// TwinCAT 3 PLC project MAS418_PLC
// ProgramVersion: 3.1.4023.0
// libraries:
//   Tc2_Standard, * (Beckhoff Automation GmbH)
//   Tc2_System, * (Beckhoff Automation GmbH)
//   Tc3_Module, * (Beckhoff Automation GmbH)
// project tree:
//   / GlobalTextList.TcGTLO, PlcTask.TcTTO, Visualization Manager.TcVMO (not stored)
//   POUs/ MAIN.TcPOU
//   VISUs/ HMI.TcVIS
// real-time tasks:
//   TASK PlcTask: cycle T#10ms, priority 20, ADS port 350

CONFIGURATION MAS418_PLC
    RESOURCE PLC ON TwinCAT3
        TASK PlcTask(INTERVAL := T#10ms, PRIORITY := 20);
        PROGRAM MAIN WITH PlcTask : MAIN;
    END_RESOURCE
END_CONFIGURATION

// ---- POUs/MAIN.TcPOU
PROGRAM MAIN
VAR
	bEnable : BOOL;
	bStart : BOOL;
	nINT : INT := -32768;
	nUINT : UINT := 65535;
	fREAL : REAL := 255.255;
END_VAR

bEnable := bStart;

END_PROGRAM

// ---- GlobalTextList.TcGTLO
TEXTLIST GlobalTextList
  775 = 'BOOL'
  109 = 'BOOL%i'
  173 = 'DataTypeTesting'
  74 = 'INT'
  710 = 'INT%i'
  986 = 'Power ON'
  573 = 'REAL'
  369 = 'REAL%i'
  65 = 'STRING'
  563 = 'STRING%i'
  393 = 'UINT'
  128 = 'UINT%i'
END_TEXTLIST

// ---- VISUs/HMI.TcVIS
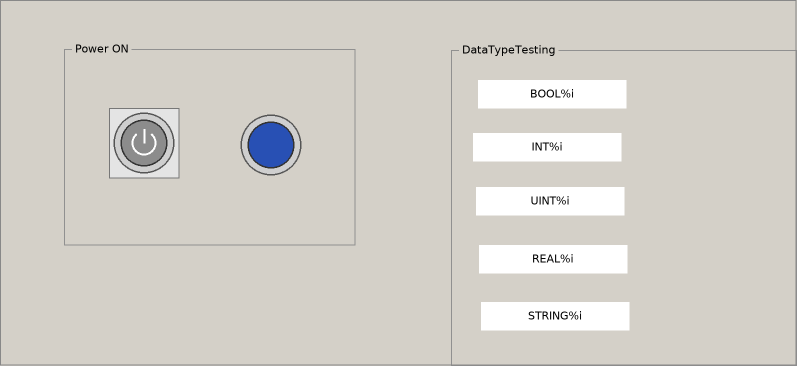
VISUALIZATION HMI  // 797x366
    GroupBox (64,41 291x204), "Power ON"
        PowerSwitch (45,67 70x70), variable: MAIN.bStart, behaviour: TOGGLE, style: Switch-PowerSwitch-Gray
        Lamp1 (172,69 70x70), variable: MAIN.bEnable, style: Lamp-Lamp1-Blue
    GroupBox (451,42 346x324), "DataTypeTesting"
        Textfield (26,37 150x30), "BOOL%i", text variable: MAIN.bEnable
        Textfield (21,90 150x30), "INT%i", text variable: MAIN.nINT
        Textfield (24,144 150x30), "UINT%i", text variable: MAIN.nUINT
        Textfield (27,202 150x30), "REAL%i", text variable: MAIN.fREAL
        Textfield (29,259 150x30), "STRING%i"
END_VISUALIZATION
